(* CODESYS project tricodrisse_projetV1.project
   Title: M241-ILS2K
   Version: 0.0.0.0
   Author: Philippe

Project tree, tasks and I/O mapping:
  MyController : TM241CE40R, Schneider Electric, order no. TM241CE40R, version 5.1.9.44
      settings: default options for OPCUA.Revision of the configuration for the stack = 2.0; default options for OPCUA.Maximum selectable variables = 2000
    application Application
      libraries: Integrated Lexium Library, 3.2.1.0 (Schneider Electric)
      task MAST (cyclic, interval 20 ms, priority 25, watchdog 200 ms x 2) calls UPDATE_COMMAND, MAIN_SFC, ILE_functionblocks
      global variables GVL
      visualisation Visualization
      program ILE_functionblocks [FBD]
      program MAIN_SFC [SFC]
      visualisation Visualization_1
      program UPDATE_COMMAND [SFC]
      program asserv [ST]
      program init [SFC]
      program UPDATE_COMMAND_1 [SFC]
      program UPDATE_COMMAND_2 [SFC]
    DI : Digital Inputs, Schneider Electric, version 5.1.9.44
        input  idwDI_IDW0 : DWORD  // IDW0
        input  ibDI_IB2 : BYTE  // IB1
    DQ : Digital Outputs, Schneider Electric, version 5.1.9.44
        output qwDQ_QW0 : WORD  // QW0
        output qbDQ_QB2 : BYTE  // QB1
    Counters : Counters, Schneider Electric, version 5.1.9.44
    Pulse_Generators : Pulse Generators, Schneider Electric, version 5.1.9.44
    Cartridge_1 : Cartridge, Schneider Electric, version 5.1.9.44
    Cartridge_2 : Cartridge, Schneider Electric, version 5.1.9.44
    IO_Bus : IO bus - TM3, Schneider Electric, version 5.1.9.44
    COM_Bus : COM bus, Schneider Electric, version 5.1.9.44
    Ethernet_1 : Ethernet Network, Schneider Electric, version 5.1.9.44
        settings: IPAddress = [292, 268, 200, 200]; SubnetMask = [255, 255, 255, 0]; GatewayAddress = [292, 268, 200, 254]; WebServer = TRUE; FTP Server = TRUE; SoMachine Protocol = TRUE; Modbus Server = TRUE; NetManage Protocol = TRUE; SNMP protocol = TRUE; Enable Routing = FALSE; WebVisu protocol = TRUE; Maximum EiP connections = 26; DHCP Server Active = TRUE; Secured Web Server = TRUE; MACAddress = [26#0, 26#0, 26#0, 26#0, 26#0, 26#0]
      Gestionnaire_Ethernet_Industriel : Industrial Ethernet Manager, Schneider Electric, version 1.0.12.40
          settings: EIP Load with penality = 200; Max devices under scanner = 228; Max connections with eip and modbus = 26; IPAddress = [292,268,0,2]; TCPFlags = 2043; Vendor Code = 2285; Product Type = 22; Product Code = 200; Major Revision = 2; Minor Revision = 2; Serial Number = 26#00000825; BinaryFileSize = 1048; unconnected timeout for explicit message = 20000; max Input assembly size = 220; max output assembly size = 220; Dhcps Host 1.Client Mac Address = [00,00,00,00,00,00]; Dhcps Host 1.Client Device Name = 'Lexium-ILx-002'; Dhcps Host 1.Client IP Address = [292, 268, 200, 202]; Dhcps Host 1.Network Mask = [255, 255, 255, 0]; Dhcps Host 1.Default Gateway = [292, 268, 200, 200]; Dhcps Host 3.Client Mac Address = [26#0, 26#0, 26#0, 26#0, 26#0]; Dhcps Host 4.Client Mac Address = [26#0, 26#0, 26#0, 26#0, 26#0]; Dhcps Host 5.Client Mac Address = [26#0, 26#0, 26#0, 26#0, 26#0]; Dhcps Host 6.Client Mac Address = [26#0, 26#0, 26#0, 26#0, 26#0]; Dhcps Host 7.Client Mac Address = [26#0, 26#0, 26#0, 26#0, 26#0]; Dhcps Host 8.Client Mac Address = [26#0, 26#0, 26#0, 26#0, 26#0]; Dhcps Host 9.Client Mac Address = [26#0, 26#0, 26#0, 26#0, 26#0]; Dhcps Host 10.Client Mac Address = [26#0, 26#0, 26#0, 26#0, 26#0]; Dhcps Host 11.Client Mac Address = [26#0, 26#0, 26#0, 26#0, 26#0]; Dhcps Host 12.Client Mac Address = [26#0, 26#0, 26#0, 26#0, 26#0]; Dhcps Host 13.Client Mac Address = [26#0, 26#0, 26#0, 26#0, 26#0]; Dhcps Host 14.Client Mac Address = [26#0, 26#0, 26#0, 26#0, 26#0]; Dhcps Host 15.Client Mac Address = [26#0, 26#0, 26#0, 26#0, 26#0]; Dhcps Host 16.Client Mac Address = [26#0, 26#0, 26#0, 26#0, 26#0]; Dhcps Host 17.Client Mac Address = [26#0, 26#0, 26#0, 26#0, 26#0]; Dhcps Host 18.Client Mac Address = [26#0, 26#0, 26#0, 26#0, 26#0]; Dhcps Host 19.Client Mac Address = [26#0, 26#0, 26#0, 26#0, 26#0]; Dhcps Host 20.Client Mac Address = [26#0, 26#0, 26#0, 26#0, 26#0]; Dhcps Host 21.Client Mac Address = [26#0, 26#0, 26#0, 26#0, 26#0]; Dhcps Host 22.Client Mac Address = [26#0, 26#0, 26#0, 26#0, 26#0];
            Dhcps Host 23.Client Mac Address = [26#0, 26#0, 26#0, 26#0, 26#0]; Dhcps Host 24.Client Mac Address = [26#0, 26#0, 26#0, 26#0, 26#0]; Dhcps Host 25.Client Mac Address = [26#0, 26#0, 26#0, 26#0, 26#0]; Dhcps Host 26.Client Mac Address = [26#0, 26#0, 26#0, 26#0, 26#0]; Dhcps Host 27.Client Mac Address = [26#0, 26#0, 26#0, 26#0, 26#0]; Dhcps Host 28.Client Mac Address = [26#0, 26#0, 26#0, 26#0, 26#0]; Dhcps Host 29.Client Mac Address = [26#0, 26#0, 26#0, 26#0, 26#0]; Dhcps Host 30.Client Mac Address = [26#0, 26#0, 26#0, 26#0, 26#0]; Dhcps Host 31.Client Mac Address = [26#0, 26#0, 26#0, 26#0, 26#0]; Dhcps Host 32.Client Mac Address = [26#0, 26#0, 26#0, 26#0, 26#0]; Dhcps Host 33.Client Mac Address = [26#0, 26#0, 26#0, 26#0, 26#0]; Dhcps Host 34.Client Mac Address = [26#0, 26#0, 26#0, 26#0, 26#0]; Dhcps Host 35.Client Mac Address = [26#0, 26#0, 26#0, 26#0, 26#0]; Dhcps Host 36.Client Mac Address = [26#0, 26#0, 26#0, 26#0, 26#0]; Dhcps Host 37.Client Mac Address = [26#0, 26#0, 26#0, 26#0, 26#0]; Dhcps Host 38.Client Mac Address = [26#0, 26#0, 26#0, 26#0, 26#0]; Dhcps Host 39.Client Mac Address = [26#0, 26#0, 26#0, 26#0, 26#0]; Dhcps Host 40.Client Mac Address = [26#0, 26#0, 26#0, 26#0, 26#0]; Dhcps Host 41.Client Mac Address = [26#0, 26#0, 26#0, 26#0, 26#0]; Dhcps Host 42.Client Mac Address = [26#0, 26#0, 26#0, 26#0, 26#0]; Dhcps Host 43.Client Mac Address = [26#0, 26#0, 26#0, 26#0, 26#0]; Dhcps Host 44.Client Mac Address = [26#0, 26#0, 26#0, 26#0, 26#0]; Dhcps Host 45.Client Mac Address = [26#0, 26#0, 26#0, 26#0, 26#0]; Dhcps Host 46.Client Mac Address = [26#0, 26#0, 26#0, 26#0, 26#0]; Dhcps Host 47.Client Mac Address = [26#0, 26#0, 26#0, 26#0, 26#0]; Dhcps Host 48.Client Mac Address = [26#0, 26#0, 26#0, 26#0, 26#0]; Dhcps Host 49.Client Mac Address = [26#0, 26#0, 26#0, 26#0, 26#0]; Dhcps Host 50.Client Mac Address = [26#0, 26#0, 26#0, 26#0, 26#0]; Dhcps Host 51.Client Mac Address = [26#0, 26#0, 26#0, 26#0, 26#0]; Dhcps Host 52.Client Mac Address = [26#0, 26#0, 26#0, 26#0, 26#0]; Dhcps Host 53.Client Mac Address = [26#0, 26#0, 26#0, 26#0, 26#0]; Dhcps Host 54.Client Mac Address = [26#0, 26#0, 26#0, 26#0, 26#0]; Dhcps Host 55.Client Mac Address = [26#0, 26#0, 26#0, 26#0, 26#0]; Dhcps Host 56.Client Mac Address = [26#0, 26#0, 26#0, 26#0, 26#0]; Dhcps Host 57.Client Mac Address = [26#0, 26#0, 26#0, 26#0, 26#0]; Dhcps Host 58.Client Mac Address = [26#0, 26#0, 26#0, 26#0, 26#0]; Dhcps Host 59.Client Mac Address = [26#0, 26#0, 26#0, 26#0, 26#0]; Dhcps Host 60.Client Mac Address = [26#0, 26#0, 26#0, 26#0, 26#0]; Dhcps Host 61.Client Mac Address = [26#0, 26#0, 26#0, 26#0, 26#0]; Dhcps Host 62.Client Mac Address = [26#0, 26#0, 26#0, 26#0, 26#0];
            Dhcps Host 63.Client Mac Address = [26#0, 26#0, 26#0, 26#0, 26#0]; Dhcps Host 64.Client Mac Address = [26#0, 26#0, 26#0, 26#0, 26#0]; Dhcps Host 65.Client Mac Address = [26#0, 26#0, 26#0, 26#0, 26#0]; Dhcps Host 66.Client Mac Address = [26#0, 26#0, 26#0, 26#0, 26#0]; Dhcps Host 67.Client Mac Address = [26#0, 26#0, 26#0, 26#0, 26#0]; Dhcps Host 68.Client Mac Address = [26#0, 26#0, 26#0, 26#0, 26#0]; Dhcps Host 69.Client Mac Address = [26#0, 26#0, 26#0, 26#0, 26#0]; Dhcps Host 70.Client Mac Address = [26#0, 26#0, 26#0, 26#0, 26#0]; Dhcps Host 71.Client Mac Address = [26#0, 26#0, 26#0, 26#0, 26#0]; Dhcps Host 72.Client Mac Address = [26#0, 26#0, 26#0, 26#0, 26#0]; Dhcps Host 73.Client Mac Address = [26#0, 26#0, 26#0, 26#0, 26#0]; Dhcps Host 74.Client Mac Address = [26#0, 26#0, 26#0, 26#0, 26#0]; Dhcps Host 75.Client Mac Address = [26#0, 26#0, 26#0, 26#0, 26#0]; Dhcps Host 76.Client Mac Address = [26#0, 26#0, 26#0, 26#0, 26#0]; Dhcps Host 77.Client Mac Address = [26#0, 26#0, 26#0, 26#0, 26#0]; Dhcps Host 78.Client Mac Address = [26#0, 26#0, 26#0, 26#0, 26#0]; Dhcps Host 79.Client Mac Address = [26#0, 26#0, 26#0, 26#0, 26#0]; Dhcps Host 80.Client Mac Address = [26#0, 26#0, 26#0, 26#0, 26#0]; Dhcps Host 81.Client Mac Address = [26#0, 26#0, 26#0, 26#0, 26#0]; Dhcps Host 82.Client Mac Address = [26#0, 26#0, 26#0, 26#0, 26#0]; Dhcps Host 83.Client Mac Address = [26#0, 26#0, 26#0, 26#0, 26#0]; Dhcps Host 84.Client Mac Address = [26#0, 26#0, 26#0, 26#0, 26#0]; Dhcps Host 85.Client Mac Address = [26#0, 26#0, 26#0, 26#0, 26#0]; Dhcps Host 86.Client Mac Address = [26#0, 26#0, 26#0, 26#0, 26#0]; Dhcps Host 87.Client Mac Address = [26#0, 26#0, 26#0, 26#0, 26#0]; Dhcps Host 88.Client Mac Address = [26#0, 26#0, 26#0, 26#0, 26#0]; Dhcps Host 89.Client Mac Address = [26#0, 26#0, 26#0, 26#0, 26#0]; Dhcps Host 90.Client Mac Address = [26#0, 26#0, 26#0, 26#0, 26#0]; Dhcps Host 91.Client Mac Address = [26#0, 26#0, 26#0, 26#0, 26#0]; Dhcps Host 92.Client Mac Address = [26#0, 26#0, 26#0, 26#0, 26#0]; Dhcps Host 93.Client Mac Address = [26#0, 26#0, 26#0, 26#0, 26#0]; Dhcps Host 94.Client Mac Address = [26#0, 26#0, 26#0, 26#0, 26#0]; Dhcps Host 95.Client Mac Address = [26#0, 26#0, 26#0, 26#0, 26#0]; Dhcps Host 96.Client Mac Address = [26#0, 26#0, 26#0, 26#0, 26#0]; Dhcps Host 97.Client Mac Address = [26#0, 26#0, 26#0, 26#0, 26#0]; Dhcps Host 98.Client Mac Address = [26#0, 26#0, 26#0, 26#0, 26#0]; Dhcps Host 99.Client Mac Address = [26#0, 26#0, 26#0, 26#0, 26#0]; Dhcps Host 100.Client Mac Address = [26#0, 26#0, 26#0, 26#0, 26#0]; Dhcps Host 101.Client Mac Address = [26#0, 26#0, 26#0, 26#0, 26#0]; Dhcps Host 102.Client Mac Address = [26#0, 26#0, 26#0, 26#0, 26#0];
            Dhcps Host 103.Client Mac Address = [26#0, 26#0, 26#0, 26#0, 26#0]; Dhcps Host 104.Client Mac Address = [26#0, 26#0, 26#0, 26#0, 26#0]; Dhcps Host 105.Client Mac Address = [26#0, 26#0, 26#0, 26#0, 26#0]; Dhcps Host 106.Client Mac Address = [26#0, 26#0, 26#0, 26#0, 26#0]; Dhcps Host 107.Client Mac Address = [26#0, 26#0, 26#0, 26#0, 26#0]; Dhcps Host 108.Client Mac Address = [26#0, 26#0, 26#0, 26#0, 26#0]; Dhcps Host 109.Client Mac Address = [26#0, 26#0, 26#0, 26#0, 26#0]; Dhcps Host 110.Client Mac Address = [26#0, 26#0, 26#0, 26#0, 26#0]; Dhcps Host 111.Client Mac Address = [26#0, 26#0, 26#0, 26#0, 26#0]; Dhcps Host 112.Client Mac Address = [26#0, 26#0, 26#0, 26#0, 26#0]; Dhcps Host 113.Client Mac Address = [26#0, 26#0, 26#0, 26#0, 26#0]; Dhcps Host 114.Client Mac Address = [26#0, 26#0, 26#0, 26#0, 26#0]; Dhcps Host 115.Client Mac Address = [26#0, 26#0, 26#0, 26#0, 26#0]; Dhcps Host 116.Client Mac Address = [26#0, 26#0, 26#0, 26#0, 26#0]; Dhcps Host 117.Client Mac Address = [26#0, 26#0, 26#0, 26#0, 26#0]; Dhcps Host 118.Client Mac Address = [26#0, 26#0, 26#0, 26#0, 26#0]; Dhcps Host 119.Client Mac Address = [26#0, 26#0, 26#0, 26#0, 26#0]; Dhcps Host 120.Client Mac Address = [26#0, 26#0, 26#0, 26#0, 26#0]; Dhcps Host 121.Client Mac Address = [26#0, 26#0, 26#0, 26#0, 26#0]; Dhcps Host 122.Client Mac Address = [26#0, 26#0, 26#0, 26#0, 26#0]; Dhcps Host 123.Client Mac Address = [26#0, 26#0, 26#0, 26#0, 26#0]; Dhcps Host 124.Client Mac Address = [26#0, 26#0, 26#0, 26#0, 26#0]; Dhcps Host 125.Client Mac Address = [26#0, 26#0, 26#0, 26#0, 26#0]; Dhcps Host 126.Client Mac Address = [26#0, 26#0, 26#0, 26#0, 26#0]; Dhcps Host 127.Client Mac Address = [26#0, 26#0, 26#0, 26#0, 26#0]; Dhcps Host 128.Client Mac Address = [26#0, 26#0, 26#0, 26#0, 26#0]; InterfaceUsedByDhcpSize = 4; InterfaceUsedByDhcp = [0,0,0,0]
          unmapped channels: Global Status, Healthbit 0, Healthbit 1, Healthbit 2, Healthbit 3, Channels 0, Channels 1, %IW20 Channels 2, %IW22 Channels 3
        Lexium_ILE_1 : Lexium ILE, Schneider Electric, order no. 89330, version 1.2.11.0
            settings: IP address of Target = [292,268,200,259]; MAC address of Target = [26#00, 26#80, 26#F4, 26#7B, 26#28, 26#E2]; Major Revision = 2; Minor Revision = 2; DeviceNumber = 1; Object Input1 = [0, 312, 268500992, 257]; Object Output1 = [1, 312, 268566528, 257]; Connection Id List = [257,0,0,0,0,0,0,0]; Number of Connections = 2; Connection Settings.Connection Number = 257; Connection Settings.Requested packet intervall (µs) = 20000; Connection Settings.OT Connection Parameters = 28478; Connection Settings.TO Connection Parameters = 28474; Connection Settings.Transport Type = 2; Connection Settings.Transmission inhibit time Scanner (ms) = 20; Connection Settings.Transmission inhibit time Target (ms) = 20; Connection Settings IPCL.Requested packet intervall T-O (µs) = 20000; Connection Settings IPCL.Requested packet intervall O-T (µs) = 20000; Connection Path = [26#20,26#04,26#24,26#02,26#2C,26#67,26#2C,26#72]
            unmapped channels: %IW22 Input Read/Write IclA, Output Read/Write IclA
        Lexium_ILE_2 : Lexium ILE, Schneider Electric, order no. 89330, version 1.2.11.0
            settings: IP address of Target = [292, 268, 200, 202]; Major Revision = 2; Minor Revision = 2; DeviceNumber = 2; Object Input1 = [4, 312, 268500992, 258]; Object Output1 = [5, 312, 268566528, 258]; Connection Id List = [258,0,0,0,0,0,0,0]; Number of Connections = 2; Connection Settings.Connection Number = 258; Connection Settings.Requested packet intervall (µs) = 20000; Connection Settings.OT Connection Parameters = 28478; Connection Settings.TO Connection Parameters = 28474; Connection Settings.Transport Type = 2; Connection Settings.Transmission inhibit time Scanner (ms) = 20; Connection Settings.Transmission inhibit time Target (ms) = 20; Connection Settings IPCL.Requested packet intervall T-O (µs) = 20000; Connection Settings IPCL.Requested packet intervall O-T (µs) = 20000; Connection Path = [26#20,26#04,26#24,26#02,26#2C,26#67,26#2C,26#72]
            unmapped channels: Input Read/Write IclA, Output Read/Write IclA
    Serial_Line_1 : Serial line, Schneider Electric, version 5.1.9.44
      SoMachine_Network_Manager : Machine Expert-Network Manager, Schneider Electric, version 4.0.0.4
    Serial_Line_2 : Serial line, Schneider Electric, version 5.1.9.44
      Modbus_Manager : Modbus Manager, Schneider Electric, version 4.0.0.4
  libraries: VisuSymbols, 3.5.10.0 (System)
  text list GlobalTextList
*)

// MyController/Application/GVL

VAR_GLOBAL
	
	//MOTEUR 2
	// Power
	ILE_2_Power_Enable : BOOL := FALSE;
	ILE_2_Power_StatusOK: BOOL;
	
	// LimitSwitches
	ILE_2_LimitSwitch_Execute : BOOL;
	ILE_2_LimitSwitch_neg_disabled,ILE_2_LimitSwitch_pos_disabled : BOOL;
	 
	// Movement (target velocity)
 	ILE_2_Movement : BOOL;
 	targetVelocity_2 : DINT := 500;
	actualVelocity_2 : DINT;
	inVelocity_2 : BOOL;
	ILE_2_Position : INT;
	Torque_2 : INT;
	Set_Position_2: BOOL;
	Set_Position_2_OK:BOOL;
	
	// Error reading
	ILE_2_ReadError : BOOL := TRUE;
	ILE_2_ReadStatus : BOOL := TRUE;
	ILE_2_ReadPosition : BOOL := TRUE;
	
	ILE_2_Reset : BOOL;
	ILE_2_ResetOK : BOOL;
	
	
	
	//MOTEUR1
	// Power
	ILE_1_Power_Enable : BOOL := FALSE;
	ILE_1_Power_StatusOK: BOOL;
	
	// LimitSwitches
	ILE_1_LimitSwitch_Execute : BOOL;
	ILE_1_LimitSwitch_neg_disabled,ILE_1_LimitSwitch_pos_disabled : BOOL;
	 
	// Movement (target velocity)
 	ILE_1_Movement : BOOL;
 	targetVelocity_1 : DINT;
	actualVelocity_1 : DINT;
	inVelocity_1 : BOOL;
	ILE_1_Position : INT;
	Torque_1 : INT;
	Set_Position_1: BOOL;
	Set_Position_1_OK:BOOL;


	
	// Error reading
	ILE_1_ReadError : BOOL := TRUE;
	ILE_1_ReadStatus : BOOL := TRUE;
	ILE_1_ReadPosition : BOOL := TRUE;
	
	ILE_1_Reset : BOOL;
	ILE_1_ResetOK : BOOL;
	
	
	//TOUS MOTEURS
	ILE_LimitSwitch_disabled : BOOL;
	Init_OK: BOOL;
	StartApp_1: BOOL;
	StartApp_2: BOOL;
	StartApp : BOOL;
	Torque_Init: INT := 200;
	Position_init: INT := 1000;
	
	//Geometry
	h_triangle : REAL;
	x : REAL;
	L1 : REAL;
	L2 : REAL;
	target_x : REAL;
	init_x : REAL;
	dist : REAL;
	v_real_mobile : REAL;
	v_target_mobile : REAL;
	demi_perimetre : REAL;
	


END_VAR

VAR_GLOBAL CONSTANT
	//Geometry constant
	pi : REAL := 3.1415;
	R_tambour : REAL := 0.0575; //trouver la bonne valeur
	h_poteau : REAL := 2.0;   //mettre la bonne valeur
	v_max_mobile : REAL := 0.10;
	target_h : REAL := 0.10;
	width : REAL:= 2.0;
	
	//moteurs
	n_point : INT := 16000;
END_VAR

// MyController/Application/UPDATE_COMMAND
PROGRAM UPDATE_COMMAND
VAR
END_VAR

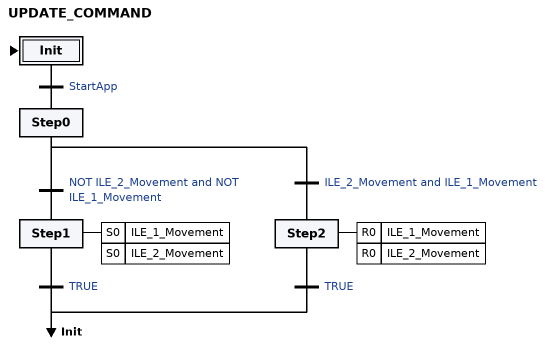
INITIAL_STEP Init:
END_STEP
TRANSITION FROM Init TO Step0
    := StartApp;
END_TRANSITION
STEP Step0:
END_STEP
TRANSITION FROM Step0 TO Step1
    := NOT ILE_2_Movement and NOT ILE_1_Movement;
END_TRANSITION
STEP Step1:
    ILE_1_Movement(S0);
    ILE_2_Movement(S0);
END_STEP
TRANSITION FROM Step1 TO Init
    := TRUE;
END_TRANSITION
TRANSITION FROM Step0 TO Step2
    := ILE_2_Movement and ILE_1_Movement;
END_TRANSITION
STEP Step2:
    ILE_1_Movement(R0);
    ILE_2_Movement(R0);
END_STEP
TRANSITION FROM Step2 TO Init
    := TRUE;
END_TRANSITION

END_PROGRAM

// MyController/Application/MAIN_SFC
PROGRAM MAIN_SFC
VAR
	ILE_ManualStart: BOOL;
	Start_asserv : BOOL;
END_VAR

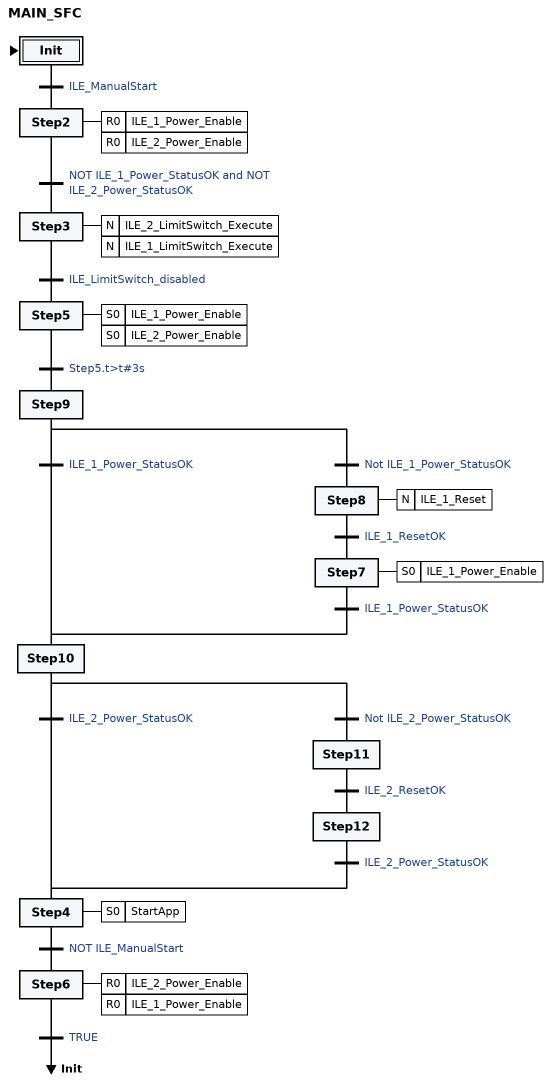
INITIAL_STEP Init:
END_STEP
TRANSITION FROM Init TO Step2
    := ILE_ManualStart;
END_TRANSITION
STEP Step2:
    ILE_1_Power_Enable(R0);
    ILE_2_Power_Enable(R0);
END_STEP
TRANSITION FROM Step2 TO Step3
    := NOT ILE_1_Power_StatusOK and NOT ILE_2_Power_StatusOK;
END_TRANSITION
STEP Step3:
    ILE_2_LimitSwitch_Execute(N);
    ILE_1_LimitSwitch_Execute(N);
END_STEP
TRANSITION FROM Step3 TO Step5
    := ILE_LimitSwitch_disabled;
END_TRANSITION
STEP Step5:
    ILE_1_Power_Enable(S0);
    ILE_2_Power_Enable(S0);
END_STEP
TRANSITION FROM Step5 TO Step9
    := Step5.t>t#3s;
END_TRANSITION
STEP Step9:
END_STEP
TRANSITION FROM Step9 TO Step10
    := ILE_1_Power_StatusOK;
END_TRANSITION
TRANSITION FROM Step9 TO Step8
    := Not ILE_1_Power_StatusOK;
END_TRANSITION
STEP Step8:
    ILE_1_Reset(N);
END_STEP
TRANSITION FROM Step8 TO Step7
    := ILE_1_ResetOK;
END_TRANSITION
STEP Step7:
    ILE_1_Power_Enable(S0);
END_STEP
TRANSITION FROM Step7 TO Step10
    := ILE_1_Power_StatusOK;
END_TRANSITION
STEP Step10:
END_STEP
TRANSITION FROM Step10 TO Step4
    := ILE_2_Power_StatusOK;
END_TRANSITION
TRANSITION FROM Step10 TO Step11
    := Not ILE_2_Power_StatusOK;
END_TRANSITION
STEP Step11:
END_STEP
TRANSITION FROM Step11 TO Step12
    := ILE_2_ResetOK;
END_TRANSITION
STEP Step12:
END_STEP
TRANSITION FROM Step12 TO Step4
    := ILE_2_Power_StatusOK;
END_TRANSITION
STEP Step4:
    StartApp(S0);
END_STEP
TRANSITION FROM Step4 TO Step6
    := NOT ILE_ManualStart;
END_TRANSITION
STEP Step6:
    ILE_2_Power_Enable(R0);
    ILE_1_Power_Enable(R0);
END_STEP
TRANSITION FROM Step6 TO Init
    := TRUE;
END_TRANSITION

END_PROGRAM

// MyController/Application/ILE_functionblocks
PROGRAM ILE_functionblocks
VAR
	MC_Power: GIPLC.MC_Power;;
	MC_ReadAxisError_2: GIPLC.MC_ReadAxisError;
	SetLimitSwitch_ILX_pos : GILXM.SetLimitSwitch_ILX;
	SetLimitSwitch_ILX_neg : GILXM.SetLimitSwitch_ILX;
	MC_ReadActualPosition: GIPLC.MC_ReadActualPosition;
	MC_ReadStatus: GIPLC.MC_ReadStatus;
	
	MC_MoveVelocity: GIPLC.MC_MoveVelocity;
	MC_Reset: GIPLC.MC_Reset;
	MC_ReadActualVelocity: GIPLC.MC_ReadActualVelocity;
	actualVelocity_2: DINT;
	MC_MoveVelocity_2: GIPLC.MC_MoveVelocity;
	MC_ReadActualVelocity_2: GIPLC.MC_ReadActualVelocity;
	inVelocity_2: BOOL;
	MC_ReadStatus_2: GIPLC.MC_ReadStatus;
	MC_ReadActualPosition_2: GIPLC.MC_ReadActualPosition;
	SetLimitSwitch_ILX_neg_2: GILXM.SetLimitSwitch_ILX;
	MC_Reset_2: GIPLC.MC_Reset;
	MC_Power_2: GIPLC.MC_Power;
	MC_ReadActualVelocity_1: GIPLC.MC_ReadActualVelocity;
	actualVelocity_1: DINT;
	MC_MoveVelocity_1: GIPLC.MC_MoveVelocity;
	inVelocity_1: BOOL;
	MC_ReadStatus_1: GIPLC.MC_ReadStatus;
	MC_ReadActualPosition_1: GIPLC.MC_ReadActualPosition;
	MC_Power_1: GIPLC.MC_Power;
	MC_Reset_1: GIPLC.MC_Reset;
	MC_ReadAxisError_1: GIPLC.MC_ReadAxisError;
	SetLimitSwitch_ILX_pos_2: GILXM.SetLimitSwitch_ILX;
	SetLimitSwitch_ILX_neg_1: GILXM.SetLimitSwitch_ILX;
	SetLimitSwitch_ILX_pos_1: GILXM.SetLimitSwitch_ILX;
	ILE_1_LimitSwitch_pos_disabled: BOOL;
	TorqueControl_LMD_0: GILXM.TorqueControl_LMD;
	TorqueControl_LMD_1: GILXM.TorqueControl_LMD;
	MC_ReadActualTorque_1: GIPLC.MC_ReadActualTorque;
	MC_ReadActualTorque_2: GIPLC.MC_ReadActualTorque;

	MC_SetPosition_1: GIPLC.MC_SetPosition;
	
	MC_SetPosition_2: GIPLC.MC_SetPosition;
END_VAR

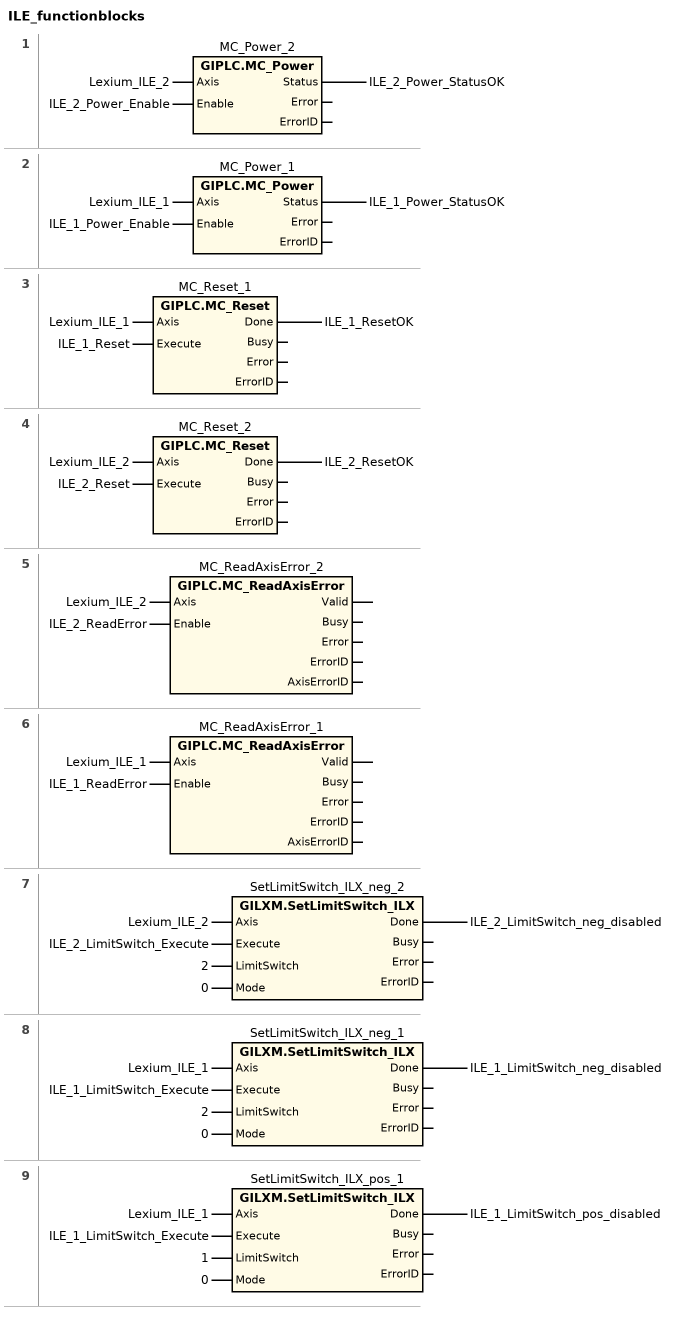
// NETWORK 1
MC_Power_2(Axis := Lexium_ILE_2, Enable := ILE_2_Power_Enable); // GIPLC.MC_Power
ILE_2_Power_StatusOK := MC_Power_2.Status;

// NETWORK 2
MC_Power_1(Axis := Lexium_ILE_1, Enable := ILE_1_Power_Enable); // GIPLC.MC_Power
ILE_1_Power_StatusOK := MC_Power_1.Status;

// NETWORK 3
MC_Reset_1(Axis := Lexium_ILE_1, Execute := ILE_1_Reset); // GIPLC.MC_Reset
ILE_1_ResetOK := MC_Reset_1.Done;

// NETWORK 4
MC_Reset_2(Axis := Lexium_ILE_2, Execute := ILE_2_Reset); // GIPLC.MC_Reset
ILE_2_ResetOK := MC_Reset_2.Done;

// NETWORK 5
MC_ReadAxisError_2(Axis := Lexium_ILE_2, Enable := ILE_2_ReadError); // GIPLC.MC_ReadAxisError

// NETWORK 6
MC_ReadAxisError_1(Axis := Lexium_ILE_1, Enable := ILE_1_ReadError); // GIPLC.MC_ReadAxisError

// NETWORK 7
SetLimitSwitch_ILX_neg_2(
    Axis := Lexium_ILE_2,
    Execute := ILE_2_LimitSwitch_Execute,
    LimitSwitch := 2,
    Mode := 0); // GILXM.SetLimitSwitch_ILX
ILE_2_LimitSwitch_neg_disabled := SetLimitSwitch_ILX_neg_2.Done;

// NETWORK 8
SetLimitSwitch_ILX_neg_1(
    Axis := Lexium_ILE_1,
    Execute := ILE_1_LimitSwitch_Execute,
    LimitSwitch := 2,
    Mode := 0); // GILXM.SetLimitSwitch_ILX
ILE_1_LimitSwitch_neg_disabled := SetLimitSwitch_ILX_neg_1.Done;

// NETWORK 9
SetLimitSwitch_ILX_pos_1(
    Axis := Lexium_ILE_1,
    Execute := ILE_1_LimitSwitch_Execute,
    LimitSwitch := 1,
    Mode := 0); // GILXM.SetLimitSwitch_ILX
ILE_1_LimitSwitch_pos_disabled := SetLimitSwitch_ILX_pos_1.Done;

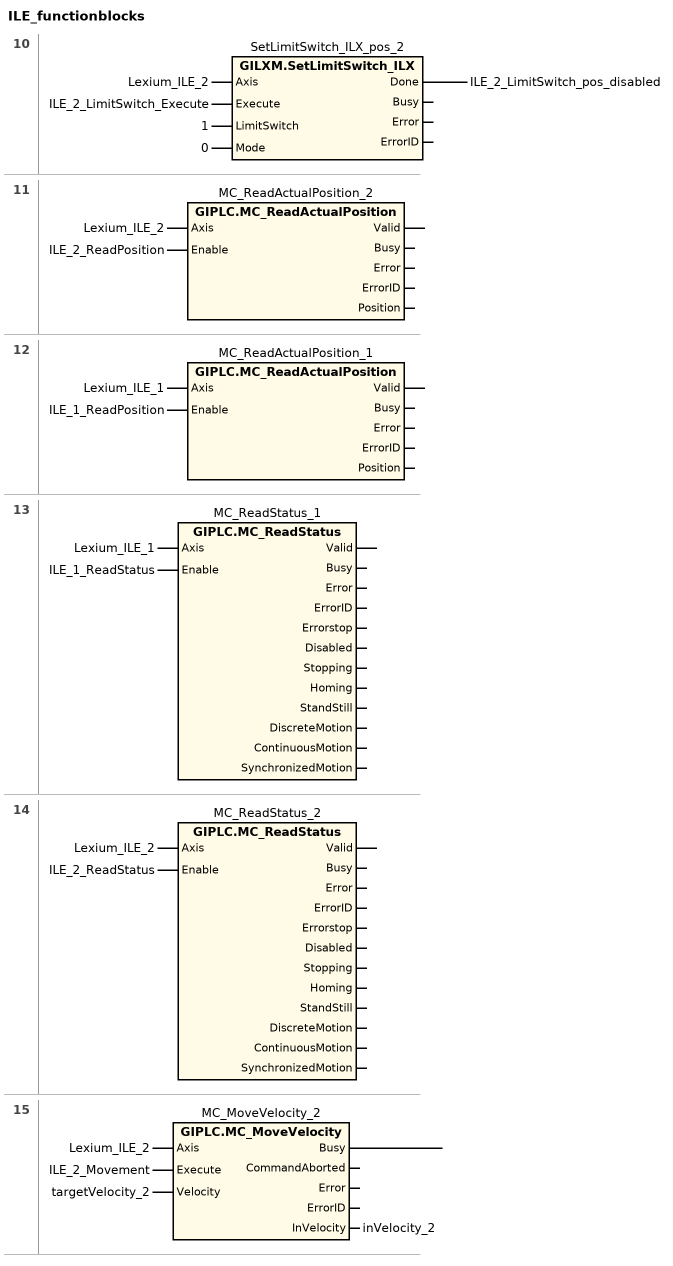
// NETWORK 10
SetLimitSwitch_ILX_pos_2(
    Axis := Lexium_ILE_2,
    Execute := ILE_2_LimitSwitch_Execute,
    LimitSwitch := 1,
    Mode := 0); // GILXM.SetLimitSwitch_ILX
ILE_2_LimitSwitch_pos_disabled := SetLimitSwitch_ILX_pos_2.Done;

// NETWORK 11
MC_ReadActualPosition_2(Axis := Lexium_ILE_2, Enable := ILE_2_ReadPosition); // GIPLC.MC_ReadActualPosition

// NETWORK 12
MC_ReadActualPosition_1(Axis := Lexium_ILE_1, Enable := ILE_1_ReadPosition); // GIPLC.MC_ReadActualPosition

// NETWORK 13
MC_ReadStatus_1(Axis := Lexium_ILE_1, Enable := ILE_1_ReadStatus); // GIPLC.MC_ReadStatus

// NETWORK 14
MC_ReadStatus_2(Axis := Lexium_ILE_2, Enable := ILE_2_ReadStatus); // GIPLC.MC_ReadStatus

// NETWORK 15
MC_MoveVelocity_2(
    Axis := Lexium_ILE_2,
    Execute := ILE_2_Movement,
    Velocity := targetVelocity_2,
    InVelocity => inVelocity_2); // GIPLC.MC_MoveVelocity

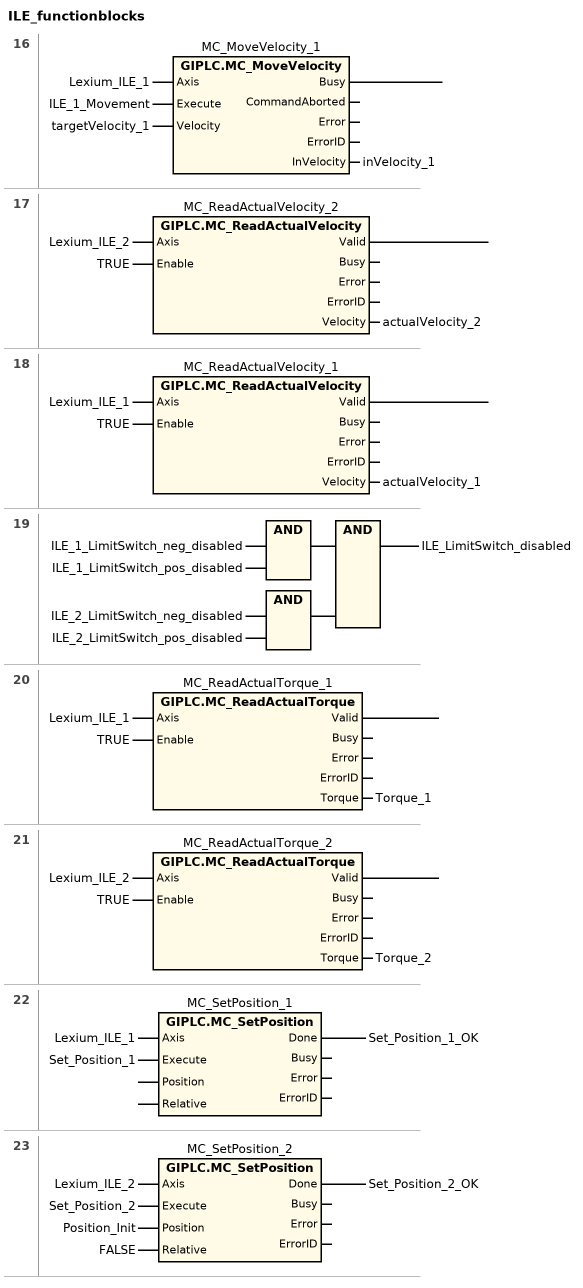
// NETWORK 16
MC_MoveVelocity_1(
    Axis := Lexium_ILE_1,
    Execute := ILE_1_Movement,
    Velocity := targetVelocity_1,
    InVelocity => inVelocity_1); // GIPLC.MC_MoveVelocity

// NETWORK 17
MC_ReadActualVelocity_2(Axis := Lexium_ILE_2, Enable := TRUE, Velocity => actualVelocity_2); // GIPLC.MC_ReadActualVelocity

// NETWORK 18
MC_ReadActualVelocity_1(Axis := Lexium_ILE_1, Enable := TRUE, Velocity => actualVelocity_1); // GIPLC.MC_ReadActualVelocity

// NETWORK 19
ILE_LimitSwitch_disabled := (ILE_1_LimitSwitch_neg_disabled AND ILE_1_LimitSwitch_pos_disabled) AND (ILE_2_LimitSwitch_neg_disabled AND ILE_2_LimitSwitch_pos_disabled);

// NETWORK 20
MC_ReadActualTorque_1(Axis := Lexium_ILE_1, Enable := TRUE, Torque => Torque_1); // GIPLC.MC_ReadActualTorque

// NETWORK 21
MC_ReadActualTorque_2(Axis := Lexium_ILE_2, Enable := TRUE, Torque => Torque_2); // GIPLC.MC_ReadActualTorque

// NETWORK 22
MC_SetPosition_1(Axis := Lexium_ILE_1, Execute := Set_Position_1); // GIPLC.MC_SetPosition
Set_Position_1_OK := MC_SetPosition_1.Done;

// NETWORK 23
MC_SetPosition_2(
    Axis := Lexium_ILE_2,
    Execute := Set_Position_2,
    Position := Position_Init,
    Relative := FALSE); // GIPLC.MC_SetPosition
Set_Position_2_OK := MC_SetPosition_2.Done;

END_PROGRAM

// MyController/Application/asserv
PROGRAM asserv
VAR
alpha : REAL; //avancement entre 0 et 1 de la trajectoire
alphadec : REAL := 0.95;
END_VAR


IF MAIN_SFC.Start_asserv = TRUE THEN

L1 := ILE_1_Position * R_tambour / n_point * 2 * pi; //attention à l'initialisation
L2 := ILE_2_Position * R_tambour / n_point * 2 * pi; //attention à l'initialisation
x := width * L1 / (L1 + L2);
demi_perimetre := (L1 + L2 + width)/2;
dist := ABS(target_x - init_x);


h_triangle := 2 / width * SQRT(demi_perimetre * (demi_perimetre - L1) * (demi_perimetre - L2) * (demi_perimetre - width)); //formule hauteur triangle
alpha := SQRT((target_x - x)*(target_x - x))/dist;
//alpha := SQRT((target_x - x)*(target_x - x) + (target_h - h)*(target_h - h))/dist;

target_h := h_poteau - h_triangle;

IF alpha <= alphadec THEN
	targetVelocity_1 := REAL_TO_INT(v_max_mobile * x / SQRT(x * x + (h_poteau - target_h) * (h_poteau - target_h)) / R_tambour / (2 * pi) * n_point);
	targetVelocity_2 := REAL_TO_INT(v_max_mobile * (x - width)/ SQRT((width - x) * (width - x) + (h_poteau - target_h) * (h_poteau - target_h)) / R_tambour / (2 * pi) * n_point);
ELSE
	//asservissement par rapport à alpha
	v_target_mobile := (1-alpha)*v_max_mobile/(1-alphadec);
	targetVelocity_1 :=  REAL_TO_INT(v_target_mobile * x / SQRT((width - x) * (width - x) + (h_poteau - target_h) * (h_poteau - target_h)) / R_tambour / (2 * pi) * n_point);
	targetVelocity_2 := REAL_TO_INT(v_target_mobile * (x - width) / SQRT((width - x) * (width - x) + (h_poteau - target_h) * (h_poteau - target_h)) / R_tambour / (2 * pi) * n_point);
END_IF


END_IF

END_PROGRAM

// MyController/Application/init
PROGRAM init
VAR
	Start_Init: BOOL;
END_VAR

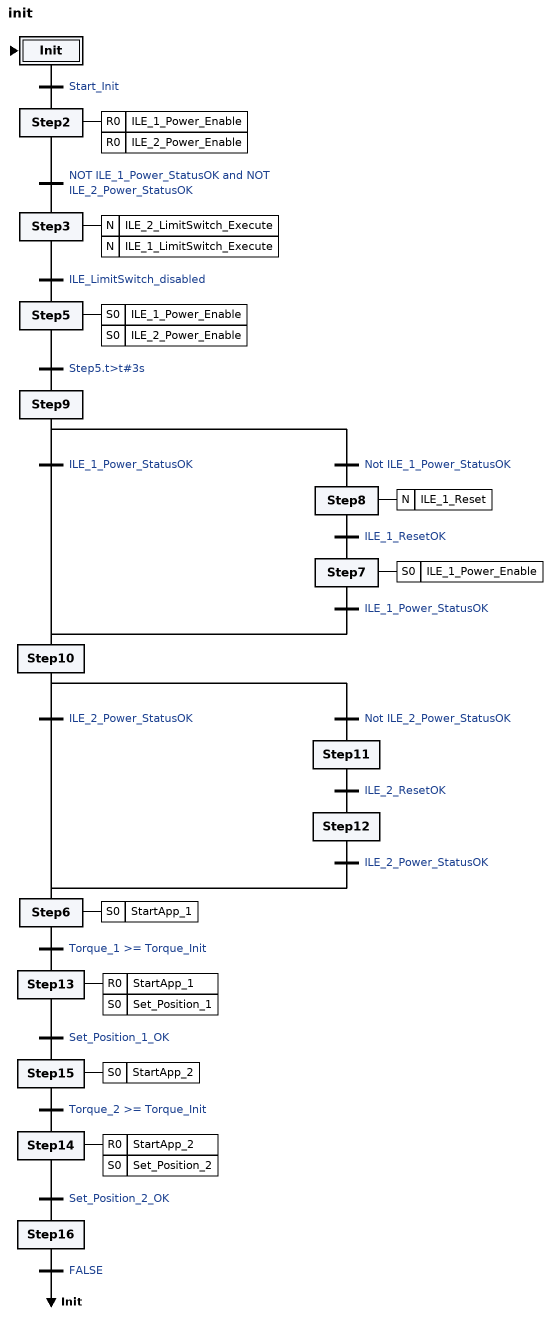
INITIAL_STEP Init:
END_STEP
TRANSITION FROM Init TO Step2
    := Start_Init;
END_TRANSITION
STEP Step2:
    ILE_1_Power_Enable(R0);
    ILE_2_Power_Enable(R0);
END_STEP
TRANSITION FROM Step2 TO Step3
    := NOT ILE_1_Power_StatusOK and NOT ILE_2_Power_StatusOK;
END_TRANSITION
STEP Step3:
    ILE_2_LimitSwitch_Execute(N);
    ILE_1_LimitSwitch_Execute(N);
END_STEP
TRANSITION FROM Step3 TO Step5
    := ILE_LimitSwitch_disabled;
END_TRANSITION
STEP Step5:
    ILE_1_Power_Enable(S0);
    ILE_2_Power_Enable(S0);
END_STEP
TRANSITION FROM Step5 TO Step9
    := Step5.t>t#3s;
END_TRANSITION
STEP Step9:
END_STEP
TRANSITION FROM Step9 TO Step10
    := ILE_1_Power_StatusOK;
END_TRANSITION
TRANSITION FROM Step9 TO Step8
    := Not ILE_1_Power_StatusOK;
END_TRANSITION
STEP Step8:
    ILE_1_Reset(N);
END_STEP
TRANSITION FROM Step8 TO Step7
    := ILE_1_ResetOK;
END_TRANSITION
STEP Step7:
    ILE_1_Power_Enable(S0);
END_STEP
TRANSITION FROM Step7 TO Step10
    := ILE_1_Power_StatusOK;
END_TRANSITION
STEP Step10:
END_STEP
TRANSITION FROM Step10 TO Step6
    := ILE_2_Power_StatusOK;
END_TRANSITION
TRANSITION FROM Step10 TO Step11
    := Not ILE_2_Power_StatusOK;
END_TRANSITION
STEP Step11:
END_STEP
TRANSITION FROM Step11 TO Step12
    := ILE_2_ResetOK;
END_TRANSITION
STEP Step12:
END_STEP
TRANSITION FROM Step12 TO Step6
    := ILE_2_Power_StatusOK;
END_TRANSITION
STEP Step6:
    StartApp_1(S0);
END_STEP
TRANSITION FROM Step6 TO Step13
    := Torque_1 >= Torque_Init;
END_TRANSITION
STEP Step13:
    StartApp_1(R0);
    Set_Position_1(S0);
END_STEP
TRANSITION FROM Step13 TO Step15
    := Set_Position_1_OK;
END_TRANSITION
STEP Step15:
    StartApp_2(S0);
END_STEP
TRANSITION FROM Step15 TO Step14
    := Torque_2 >= Torque_Init;
END_TRANSITION
STEP Step14:
    StartApp_2(R0);
    Set_Position_2(S0);
END_STEP
TRANSITION FROM Step14 TO Step16
    := Set_Position_2_OK;
END_TRANSITION
STEP Step16:
END_STEP
TRANSITION FROM Step16 TO Init
    := FALSE;
END_TRANSITION

END_PROGRAM

// MyController/Application/UPDATE_COMMAND_1
PROGRAM UPDATE_COMMAND_1
VAR
END_VAR

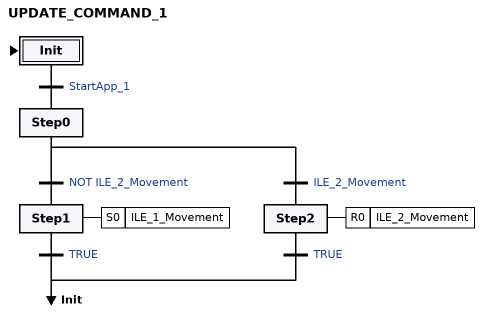
INITIAL_STEP Init:
END_STEP
TRANSITION FROM Init TO Step0
    := StartApp_1;
END_TRANSITION
STEP Step0:
END_STEP
TRANSITION FROM Step0 TO Step1
    := NOT ILE_2_Movement;
END_TRANSITION
STEP Step1:
    ILE_1_Movement(S0);
END_STEP
TRANSITION FROM Step1 TO Init
    := TRUE;
END_TRANSITION
TRANSITION FROM Step0 TO Step2
    := ILE_2_Movement;
END_TRANSITION
STEP Step2:
    ILE_2_Movement(R0);
END_STEP
TRANSITION FROM Step2 TO Init
    := TRUE;
END_TRANSITION

END_PROGRAM

// MyController/Application/UPDATE_COMMAND_2
PROGRAM UPDATE_COMMAND_2
VAR
END_VAR

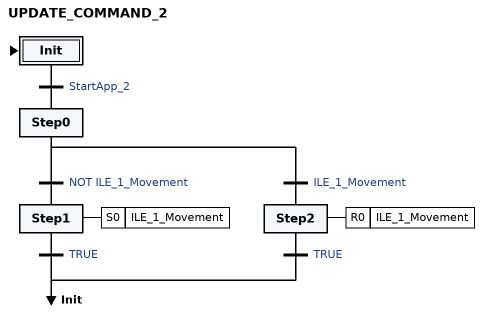
INITIAL_STEP Init:
END_STEP
TRANSITION FROM Init TO Step0
    := StartApp_2;
END_TRANSITION
STEP Step0:
END_STEP
TRANSITION FROM Step0 TO Step1
    := NOT ILE_1_Movement;
END_TRANSITION
STEP Step1:
    ILE_1_Movement(S0);
END_STEP
TRANSITION FROM Step1 TO Init
    := TRUE;
END_TRANSITION
TRANSITION FROM Step0 TO Step2
    := ILE_1_Movement;
END_TRANSITION
STEP Step2:
    ILE_1_Movement(R0);
END_STEP
TRANSITION FROM Step2 TO Init
    := TRUE;
END_TRANSITION

END_PROGRAM

// MyController/Application/Visualization
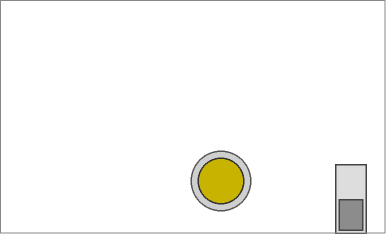
VISUALIZATION Visualization  // 386x234
    Lamp1 (186,146 70x70), variable: ILE_functionblocks.power, style: Lamp-Lamp2-Yellow
    DipSwitch (316,164 70x70), behaviour: TOGGLE, style: Switch-DipSwitch-Gray
END_VISUALIZATION

// MyController/Application/Visualization_1
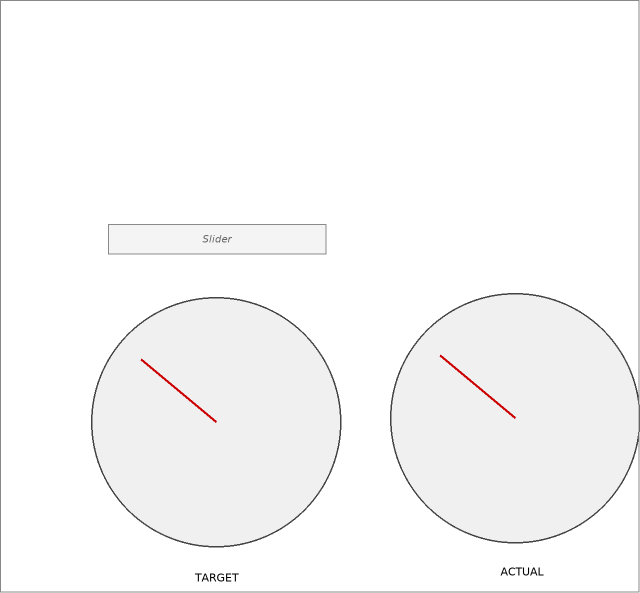
VISUALIZATION Visualization_1  // 640x593
    Slider (108,224 218x30), variable: targetVelocity, scale 0..4900
    Meter360 (390,293 250x250), value: actualVelocity, style: Meter-Meter360-Gray, scale format: %.2f, scale 0..5000
    Meter360 (91,297 250x250), value: targetVelocity, style: Meter-Meter360-Gray, scale format: %.2f, scale 0..5000
    Label (142,563 150x30), "TARGET"
    Label (447,557 150x30), "ACTUAL"
END_VISUALIZATION
